INTERFACE IPLCopenCall EXTENDS __SYSTEM.IQueryInterface

METHOD Start : PLCopenStatusBase
VAR_INPUT
  Command : IPLCopenCommand;
END_VAR
END_METHOD

END_INTERFACE

(* stored: Version 1.1.0.1
   Itf IPLCopenCall: Id {f7958e5a-b87e-0290-18b9-18a7ee86d87d}
   Method Start: Id {2089c624-b436-0a5a-1399-c3962d9edd84} *)
